{attribute 'GeneratedUsingTerminal: EL3681-0000-0021'}
{attribute addProperty BoxType "EL3681-0000-0021"}
{attribute addProperty Id "SettingsAT %I*Settings_24C049402"}
{attribute addProperty CRC "3183439273"}
{attribute addProperty Size "2"}
TYPE SAI_Feedback_BDBF6DA9 EXTENDS InputBase_8311D824 :
STRUCT
	{attribute addProperty Name "Settings"}
	Settings AT %I* : Settings_24C04940;
END_STRUCT
END_TYPE

(* stored: Version 1.2.0.0, ProductVersion 3.1.4024.11
   DUT SAI_Feedback_BDBF6DA9: Id {390e0972-f439-4070-b433-7d9d5466b937} *)
